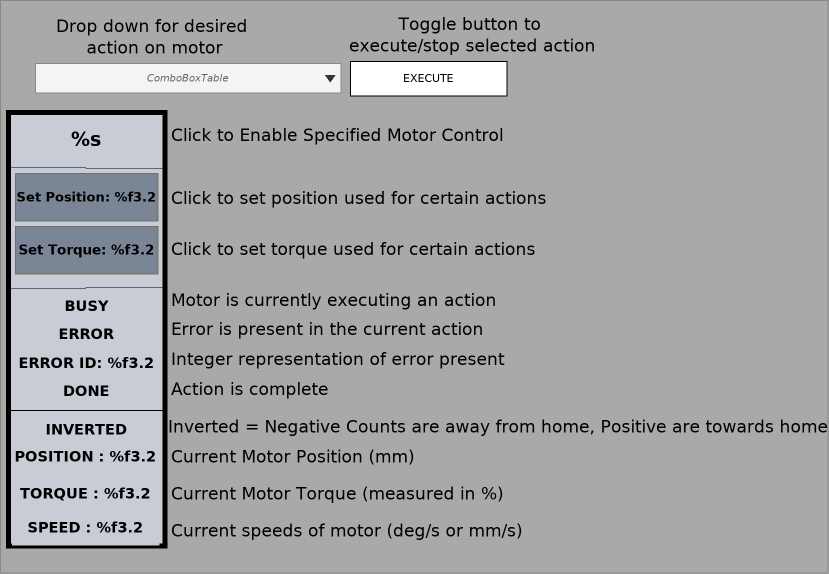
VISUALIZATION multiControlHelp  // 829x574
    Label (168,115 649x40), "Click to Enable Specified Motor Control"
    Label (168,178 649x40), "Click to set position used for certain actions"
    Label (168,229 649x40), "Click to set torque used for certain actions"
    Label (168,280 649x40), "Motor is currently executing an action"
    Label (168,309 649x40), "Error is present in the current action"
    Label (168,339 649x40), "Integer representation of error present"
    Label (168,369 649x40), "Action is complete"
    Label (168,439 649x35), "Current Motor Position (mm)"
    Label (168,476 649x35), "Current Motor Torque (measured in %)"
    Label (168,513 649x35), "Current speeds of motor (deg/s or mm/s)"
    RoundedRectangle (350,61 157x35), "EXECUTE"
    ComboBoxTable (35,63 306x30), data array: multiControl.aActionList
        p3854506369: multiControl.aActionList[INDEX]
    Rectangle (6,110 161x438)
    RoundedRectangle (14,116 145x47), "%s"
    Rectangle (12,439 147x35), "POSITION : %f3.2"
    Rectangle (15,293 143x26), "BUSY"
    Rectangle (15,378 143x26), "DONE"
    Rectangle (15,321 143x26), "ERROR"
    Rectangle (15,350 143x26), "ERROR ID: %f3.2"
    Rectangle (12,476 147x35), "TORQUE : %f3.2"
    Rectangle (12,510 147x35), "SPEED : %f3.2"
    Button (15,173 143x48), "Set Position: %f3.2"
    Button (15,226 143x48), "Set Torque: %f3.2"
    Line (6,167) (165,168)
    Line (6,288) (165,287)
    Line (6,410) (167,410)
    Label (39,16 231x42), "Drop down for desired action on motor"
    Label (350,11 245x48), "Toggle button to execute/stop selected action"
    Rectangle (15,413 143x33), "INVERTED"
    Label (165,409 663x35), "Inverted = Negative Counts are away from home, Positive are towards home."
END_VISUALIZATION

(* stored: Version 1.1.0.1, ProductVersion 3.1.4024.13
   Visu multiControlHelp: Id {22c0eb6a-6a2c-4a8e-9c1b-337fe36c235a} *)
